% RSLogix 500 project Pressure Receiver Pump Control & Indicator Logic.RSS, saved by version 8.30.00.16 %
PROJECT "PROJ11"    % processor: Bul.1763 MicroLogix 1100 Series B %

PROGRAM FILES
  LAD 2 "MAIN"  3 rungs
  LAD 3 "DIGITAL IO"  5 rungs
  LAD 4 "CONTROLS"  4 rungs

DATA FILES
  O0 OUTPUT  5 elements
  I1 INPUT  7 elements
  S2 STATUS  66 elements
  B3 BINARY  1 elements
  T4 TIMER  1 elements
  C5 COUNTER  1 elements
  R6 CONTROL  1 elements
  N7 INTEGER  1 elements
  F8 FLOAT  1 elements

LADDER 2 "MAIN"
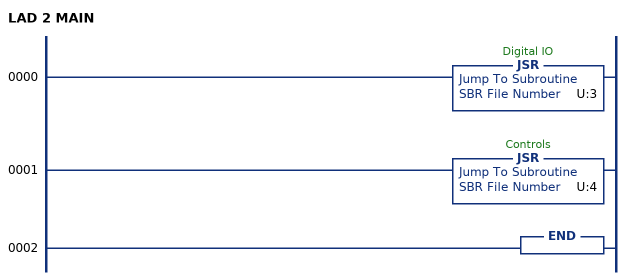
% Rung: 0 %  % edit flag set %
SOR JSR U:3 EOR
%   U:3  "Digital IO" %
% Rung: 1 %  % edit flag set %
SOR JSR U:4 EOR
%   U:4  "Controls" %
% Rung: 2 %
SOR END EOR

LADDER 3 "DIGITAL IO"
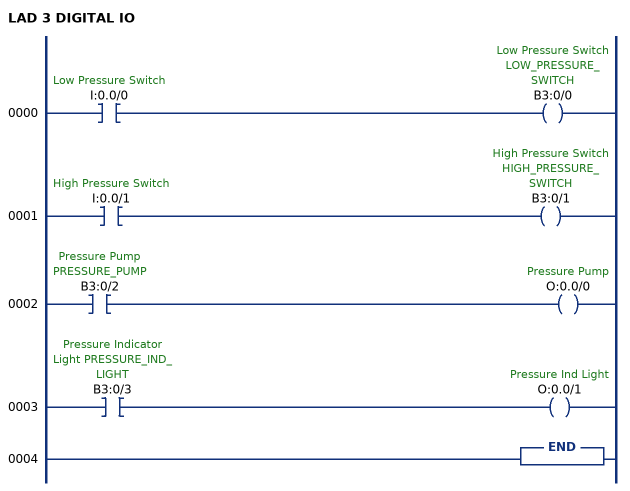
% Rung: 0 %  % edit flag set %
SOR XIC I:0.0/0 OTE B3:0/0 EOR
%   I:0.0/0  "Low Pressure Switch" %
%   B3:0/0  LOW_PRESSURE_SWITCH  "Low Pressure Switch" %
% Rung: 1 %  % edit flag set %
SOR XIC I:0.0/1 OTE B3:0/1 EOR
%   I:0.0/1  "High Pressure Switch" %
%   B3:0/1  HIGH_PRESSURE_SWITCH  "High Pressure Switch" %
% Rung: 2 %  % edit flag set %
SOR XIC B3:0/2 OTE O:0.0/0 EOR
%   B3:0/2  PRESSURE_PUMP  "Pressure Pump" %
%   O:0.0/0  "Pressure Pump" %
% Rung: 3 %  % edit flag set %
SOR XIC B3:0/3 OTE O:0.0/1 EOR
%   B3:0/3  PRESSURE_IND_LIGHT  "Pressure Indicator Light" %
%   O:0.0/1  "Pressure Ind Light" %
% Rung: 4 %
SOR END EOR

LADDER 4 "CONTROLS"
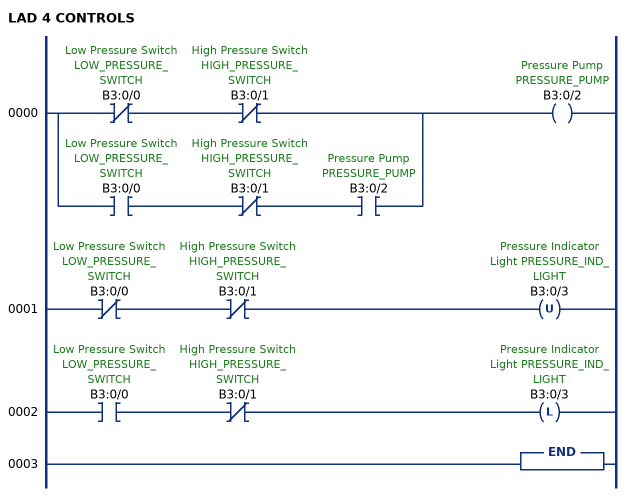
% Rung: 0 %  % edit flag set %
SOR BST XIO B3:0/0 XIO B3:0/1 NXB XIC B3:0/0 XIO B3:0/1 XIC B3:0/2 BND OTE B3:0/2 EOR
%   B3:0/0  LOW_PRESSURE_SWITCH  "Low Pressure Switch" %
%   B3:0/1  HIGH_PRESSURE_SWITCH  "High Pressure Switch" %
%   B3:0/2  PRESSURE_PUMP  "Pressure Pump" %
% Rung: 1 %  % edit flag set %
SOR XIO B3:0/0 XIO B3:0/1 OTU B3:0/3 EOR
%   B3:0/0  LOW_PRESSURE_SWITCH  "Low Pressure Switch" %
%   B3:0/1  HIGH_PRESSURE_SWITCH  "High Pressure Switch" %
%   B3:0/3  PRESSURE_IND_LIGHT  "Pressure Indicator Light" %
% Rung: 2 %  % edit flag set %
SOR XIC B3:0/0 XIO B3:0/1 OTL B3:0/3 EOR
%   B3:0/0  LOW_PRESSURE_SWITCH  "Low Pressure Switch" %
%   B3:0/1  HIGH_PRESSURE_SWITCH  "High Pressure Switch" %
%   B3:0/3  PRESSURE_IND_LIGHT  "Pressure Indicator Light" %
% Rung: 3 %
SOR END EOR
